FUNCTION_BLOCK FB_Ambient
VAR_INPUT
END_VAR
VAR_OUTPUT
	{attribute 'OPC.UA.DA' := '1'}
	localState : ST_AmbientState;
END_VAR
VAR
	WeatherStation : FB_WeatherStation;
	AmbientTemperatureSensor_Container : FB_TemperatureSensor_KL3214;
	HallTemperatureSensor_Section1 : FB_TemperatureSensor;
	HallTemperatureSensor_Section2 : FB_TemperatureSensor;
	HallTemperatureSensor_Section3 : FB_TemperatureSensor;
END_VAR

WeatherStation();
HallTemperatureSensor_Section1();
HallTemperatureSensor_Section1.GetState_AI();
HallTemperatureSensor_Section2();
HallTemperatureSensor_Section2.GetState_AI();
HallTemperatureSensor_Section3();
HallTemperatureSensor_Section3.GetState_AI();
AmbientTemperatureSensor_Container();
AmbientTemperatureSensor_Container.GetState_AI();

//add ambient temperature rain etc. from weather station
localState.fOutsideTemperature_Container := AmbientTemperatureSensor_Container.fTemperature;
localState.fOutsideTemperature := WeatherStation.fTemperature;
localState.fOutsideTemperature_Mean := WeatherStation.fMeanTemperature;
localState.bRain := WeatherStation.bRain;
localState.fDawn := WeatherStation.fDawn;
localState.fWindSpeed := WeatherStation.fWindSpeed;
localState.fHallTemperature := HallTemperatureSensor_Section3.fTemperature;

END_FUNCTION_BLOCK

(* stored: Version 1.1.0.1, ProductVersion 3.1.4024.10
   POU FB_Ambient: Id {e5737b3d-b420-44a4-9ae1-301270e5edfa}, SpecialFunc None *)
